Fanuc TP program (LS listing): calib_2.ls

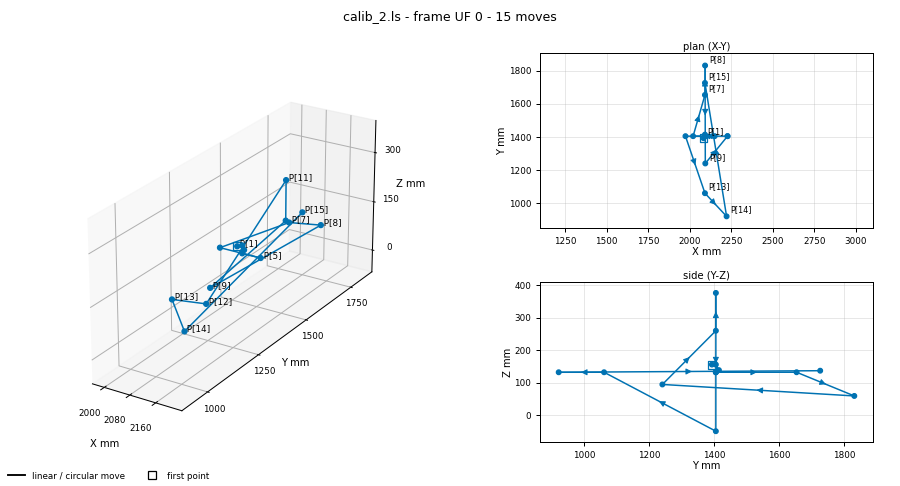
[picture p0: tool path of calib_2.ls in frame UF 0, 15 of 15 moves have a stored position in this frame; points joined in program order, loops and branches not executed]
/PROG  CALIB_2
/ATTR
OWNER		= MNEDITOR;
COMMENT		= "";
PROG_SIZE	= 1579;
CREATE		= DATE 25-09-25  TIME 18:17:04;
MODIFIED	= DATE 25-09-25  TIME 18:17:04;
FILE_NAME	= ;
VERSION		= 0;
LINE_COUNT	= 25;
MEMORY_SIZE	= 1851;
PROTECT		= READ_WRITE;
TCD:  STACK_SIZE	= 0,
      TASK_PRIORITY	= 50,
      TIME_SLICE	= 0,
      BUSY_LAMP_OFF	= 0,
      ABORT_REQUEST	= 0,
      PAUSE_REQUEST	= 0;
DEFAULT_GROUP	= 1,1,*,*,*;
CONTROL_CODE	= 00000000 00000000;
LOCAL_REGISTERS	= 0,0,0;
/MN
   1:  UFRAME_NUM=0 ;
   2:  UTOOL_NUM=10 ;
   3:  OVERRIDE=20% ;
   4:   ;
   5:L P[1] 100mm/sec FINE    ;
   6:L P[2] 100mm/sec FINE    ;
   7:L P[3] 100mm/sec FINE    ;
   8:   ;
   9:L P[4] 100mm/sec FINE    ;
  10:L P[5] 100mm/sec FINE    ;
  11:L P[6] 100mm/sec FINE    ;
  12:   ;
  13:L P[7] 100mm/sec FINE    ;
  14:L P[8] 100mm/sec FINE    ;
  15:L P[9] 100mm/sec FINE    ;
  16:   ;
  17:L P[10] 100mm/sec FINE    ;
  18:L P[11] 100mm/sec FINE    ;
  19:L P[12] 100mm/sec FINE    ;
  20:   ;
  21:L P[13] 100mm/sec FINE    ;
  22:L P[14] 100mm/sec FINE    ;
  23:L P[15] 100mm/sec FINE    ;
  24:   ;
  25:   ;
/POS
P[1]{
   GP1:
	UF : 0, UT : 10,		CONFIG : 'N U T, 0, 0, 0',
	X =  2083.354  mm,	Y =  1393.346  mm,	Z =   156.086  mm,
	W =  -179.961 deg,	P =      .020 deg,	R =   -88.855 deg
   GP2:
	UF : 0, UT : 10,
	J1=     -.082 deg
};
P[2]{
   GP1:
	UF : 0, UT : 10,		CONFIG : 'N U T, 0, 0, 0',
	X =  2091.906  mm,	Y =  1405.372  mm,	Z =   156.040  mm,
	W =  -179.962 deg,	P =      .019 deg,	R =   -88.855 deg
   GP2:
	UF : 0, UT : 10,
	J1=     -.082 deg
};
P[3]{
   GP1:
	UF : 0, UT : 10,		CONFIG : 'N U T, 0, 0, 0',
	X =  2091.930  mm,	Y =  1414.806  mm,	Z =   139.022  mm,
	W =  -179.964 deg,	P =      .018 deg,	R =   -88.856 deg
   GP2:
	UF : 0, UT : 10,
	J1=     -.082 deg
};
P[4]{
   GP1:
	UF : 0, UT : 10,		CONFIG : 'N U T, 0, 0, 0',
	X =  2091.871  mm,	Y =  1405.419  mm,	Z =   132.603  mm,
	W =  -179.965 deg,	P =      .017 deg,	R =   -88.854 deg
   GP2:
	UF : 0, UT : 10,
	J1=     -.082 deg
};
P[5]{
   GP1:
	UF : 0, UT : 10,		CONFIG : 'N U T, 0, 0, 0',
	X =  2150.273  mm,	Y =  1405.423  mm,	Z =   132.557  mm,
	W =  -179.966 deg,	P =      .016 deg,	R =   -88.854 deg
   GP2:
	UF : 0, UT : 10,
	J1=     -.082 deg
};
P[6]{
   GP1:
	UF : 0, UT : 10,		CONFIG : 'N U T, 0, 0, 0',
	X =  2020.465  mm,	Y =  1405.391  mm,	Z =   132.507  mm,
	W =  -179.967 deg,	P =      .015 deg,	R =   -88.855 deg
   GP2:
	UF : 0, UT : 10,
	J1=     -.082 deg
};
P[7]{
   GP1:
	UF : 0, UT : 10,		CONFIG : 'N U T, 0, 0, 0',
	X =  2091.832  mm,	Y =  1653.605  mm,	Z =   132.519  mm,
	W =   179.640 deg,	P =   -18.893 deg,	R =   -88.788 deg
   GP2:
	UF : 0, UT : 10,
	J1=     -.082 deg
};
P[8]{
   GP1:
	UF : 0, UT : 10,		CONFIG : 'N U T, 0, 0, 0',
	X =  2092.658  mm,	Y =  1831.070  mm,	Z =    59.637  mm,
	W =   179.254 deg,	P =   -34.144 deg,	R =   -88.613 deg
   GP2:
	UF : 0, UT : 10,
	J1=     -.082 deg
};
P[9]{
   GP1:
	UF : 0, UT : 10,		CONFIG : 'N U T, 0, 0, 0',
	X =  2093.977  mm,	Y =  1241.042  mm,	Z =    94.975  mm,
	W =  -179.691 deg,	P =    13.725 deg,	R =   -88.820 deg
   GP2:
	UF : 0, UT : 10,
	J1=     -.082 deg
};
P[10]{
   GP1:
	UF : 0, UT : 10,		CONFIG : 'N U T, 0, 0, 0',
	X =  2227.932  mm,	Y =  1405.430  mm,	Z =   260.058  mm,
	W =   174.232 deg,	P =      .131 deg,	R =   -88.861 deg
   GP2:
	UF : 0, UT : 10,
	J1=     -.082 deg
};
P[11]{
   GP1:
	UF : 0, UT : 10,		CONFIG : 'N U T, 0, 0, 0',
	X =  2227.913  mm,	Y =  1405.476  mm,	Z =   376.311  mm,
	W =   169.254 deg,	P =      .228 deg,	R =   -88.876 deg
   GP2:
	UF : 0, UT : 10,
	J1=     -.082 deg
};
P[12]{
   GP1:
	UF : 0, UT : 10,		CONFIG : 'N U T, 0, 0, 0',
	X =  1974.451  mm,	Y =  1405.388  mm,	Z =   -48.749  mm,
	W =  -172.528 deg,	P =     -.132 deg,	R =   -88.862 deg
   GP2:
	UF : 0, UT : 10,
	J1=     -.082 deg
};
P[13]{
   GP1:
	UF : 0, UT : 10,		CONFIG : 'N U T, 0, 0, 0',
	X =  2091.843  mm,	Y =  1061.746  mm,	Z =   132.477  mm,
	W =  -179.968 deg,	P =      .015 deg,	R =   -74.727 deg
   GP2:
	UF : 0, UT : 10,
	J1=     -.082 deg
};
P[14]{
   GP1:
	UF : 0, UT : 10,		CONFIG : 'N U T, 0, 0, 0',
	X =  2222.197  mm,	Y =   922.253  mm,	Z =   132.427  mm,
	W =  -179.970 deg,	P =      .015 deg,	R =   -67.418 deg
   GP2:
	UF : 0, UT : 10,
	J1=     -.082 deg
};
P[15]{
   GP1:
	UF : 0, UT : 10,		CONFIG : 'N U T, 0, 0, 0',
	X =  2091.861  mm,	Y =  1726.193  mm,	Z =   137.228  mm,
	W =  -179.969 deg,	P =      .013 deg,	R =  -102.453 deg
   GP2:
	UF : 0, UT : 10,
	J1=     -.082 deg
};
/END
